RoboDK station: FanucComputerVisionSimulation_V1.rdk

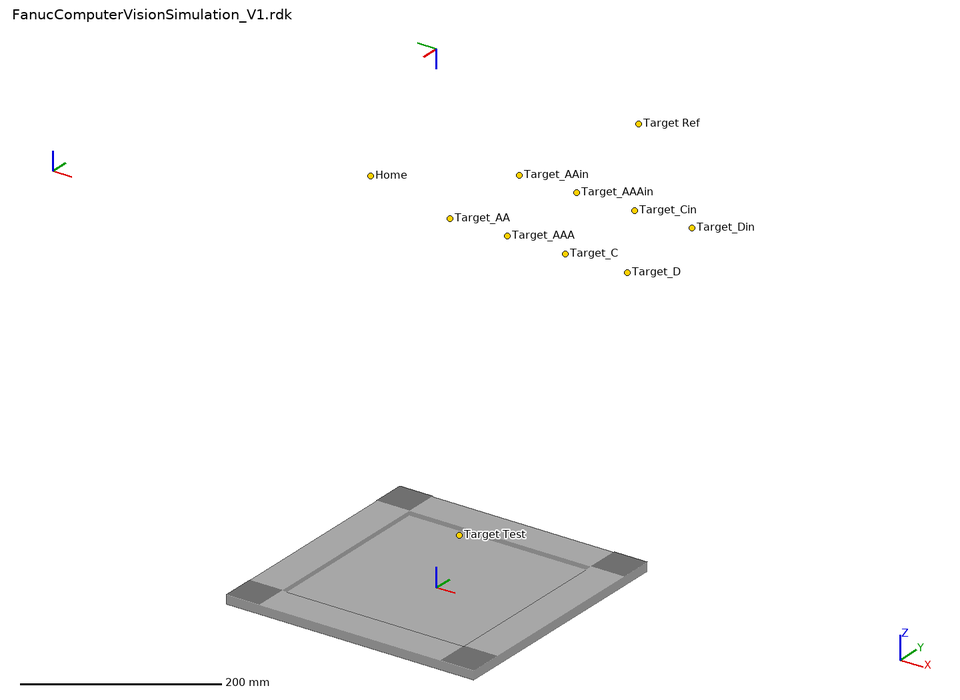
[picture v0: the station drawn from its stored meshes, robots at their saved joint values, targets as dots, program paths as lines]
Station FanucComputerVisionSimulation_V1 (saved by RoboDK 5.5.4). Poses are relative to the parent item; angles as X-Y-Z fixed-axis rotations.
Station parameters (name, value as stored): boardCenter, (319.0, 239.5, True), battery0, (496.821942952221, 61.274491474303716), battery1, (530.5798901508712, -36.737235512468814), battery2, (410.82767440352166, 59.47826360901432), battery3, (391.48109251529473, -70.56545100399168)
  - frame Fanuc LR Mate 200iD Base at (0, 0, 330) mm
    - robot Fanuc LR Mate 200iD: 6 axes, payload 7 kg, reach 717 mm, repeatability 0.02 mm, weight 25 kg
        modified DH rows (alpha deg, a mm, theta deg, d mm): 0, 0, 0, 330; -90, 50, -90, 0; 0, 330, 0, 0; -90, 35, 0, 335; 90, 0, 0, 0; -90, 0, 0, 80
        base shift (0, 0, -330) mm
        joint limits [-170, -100, -67, -190, -125, -360] to [170, 145, 213, 190, 125, 360]; home [0, 0, 0, 0, 0, 0]; saved at [0, 0, 0, 0, -90, 0]
      - frame My Camera Frame at (80, 0, 20) mm, rotated rx 0 ry 0 rz 90 deg
      - tool Gripper, TCP at (0, 0, 183) mm
    - frame Reference SW at (465, 0, -330) mm
      - object Work_Table at (0, 0, 0) mm, size 300 x 300 x 10 mm, 1061997773 curves, geometry from Flange_Holder.stl
        - object 4x4_1000-0 at (110, 110, 10.5) mm, size 40.5 x 40.5 x 0 mm, 862301904 curves, geometry from 4x4_1000-0.svg
        - object 4x4_1000-1 at (110, -150, 10.5) mm, size 40.5 x 40.5 x 0 mm, 862300704 curves, geometry from 4x4_1000-1.svg
        - object 4x4_1000-2 at (-150, -150, 10.5) mm, size 40.5 x 40.5 x 0 mm, 862301664 curves, geometry from 4x4_1000-2.svg
        - object 4x4_1000-3 at (-150, 110, 10.5) mm, size 40.5 x 40.5 x 0 mm, 862302864 curves, geometry from 4x4_1000-3.svg
      - target Home (Cartesian target) at (-80, 0, 432) mm, rotated rx -180 ry 0 rz 0 deg; joints [0, 0, 0, 0, -90, 0] of Fanuc LR Mate 200iD
      - target Target Ref (Cartesian target) at (70, 250, 432) mm, rotated rx -180 ry 0 rz 0 deg; joints [25.046, 43.834, 16.178, 0, -106.178, -25.046] of Fanuc LR Mate 200iD
      - target Target Test (Cartesian target) at (68.34, -58.43, 100) mm, rotated rx -180 ry 0 rz 0 deg; joints [7.615, 7.792, -3.745, 0, -86.255, -7.615] of Fanuc LR Mate 200iD
      - target Target_AA (Cartesian target) at (-110, 180, 305) mm, rotated rx -180 ry 0 rz 0 deg; joints [26.887, 3.808, -20.454, 0, -69.546, -26.887] of Fanuc LR Mate 200iD
      - target Target_AAA (Cartesian target) at (-40, 180, 305) mm, rotated rx -180 ry 0 rz 0 deg; joints [22.954, 14.574, -18.722, 0, -71.278, -22.954] of Fanuc LR Mate 200iD
      - target Target_C (Cartesian target) at (30, 180, 305) mm, rotated rx -180 ry 0 rz 0 deg; joints [19.983, 25.857, -14.839, 0, -75.161, -19.983] of Fanuc LR Mate 200iD
      - target Target_D (Cartesian target) at (105, 180, 305) mm, rotated rx -180 ry 0 rz 0 deg; joints [17.526, 39.754, -7.445, 0, -82.555, -17.526] of Fanuc LR Mate 200iD
      - target Target_AAin (Cartesian target) at (-110, 300, 305) mm, rotated rx -180 ry 0 rz 0 deg; joints [40.2, 15.123, -18.581, 0, -71.419, -40.2] of Fanuc LR Mate 200iD
      - target Target_AAAin (Cartesian target) at (-40, 300, 305) mm, rotated rx -180 ry 0 rz 0 deg; joints [35.218, 24.697, -15.33, 0, -74.67, -35.218] of Fanuc LR Mate 200iD
      - target Target_Cin (Cartesian target) at (30, 300, 305) mm, rotated rx -180 ry 0 rz 0 deg; joints [31.218, 35.742, -9.854, 0, -80.146, -31.218] of Fanuc LR Mate 200iD
      - target Target_Din (Cartesian target) at (100, 300, 305) mm, rotated rx -180 ry 0 rz 0 deg; joints [27.967, 50.525, 0.035, 0, -90.035, -27.967] of Fanuc LR Mate 200iD
  - Python program CameraProgram (listed below)
  - camera My Camera
  - object Table 108x114x32 IN at (-435, 0, -467.5) mm
  - Python program TakePhoto (listed below)
  - Python program SearchWorkArea (listed below)
  - Python program Test (listed below)
  - Python program CollectImages_size (listed below)
  - Python program CollectImages_brand (listed below)
  - frame Bateries at (-10000, 1500, 22) mm
    - object 9V(Duracell) at (0, 0, 0) mm
    - object 9V(Energizer) at (0, 0, 0) mm
    - object 9V(Lorem Ipsum) at (0, 0, 0) mm
    - object AA(Duracell) at (200, 0, -10) mm
    - object AA(Energizer) at (200, 80, -10) mm
    - object AA(Lorem Ipsum) at (200, 160, -10) mm
    - object AAA(Duracell) at (160, 0, -12) mm
    - object AAA(Energizer) at (160, 80, -12) mm
    - object AAA(Lorem Ipsum) at (160, 160, -12) mm
    - object C(Duracell) at (120, 0, -4) mm, size 6 x 3 x 6 mm, 1058642330 curves, geometry from C(Duracell).obj
    - object C(Energizer) at (120, 80, -4) mm, size 6 x 3 x 6 mm, 1058642330 curves, geometry from C(Energizer).obj
    - object C(Lorem Ipsum) at (120, 160, -4) mm, size 6 x 3 x 6 mm, 1058642330 curves, geometry from C(Lorem Ipsum).obj
    - object D(Duracell) at (80, 0, 0) mm, size 6 x 3 x 6 mm, 1058642330 curves, geometry from D(Duracell).obj
    - object D(Energizer) at (80, 80, 0) mm, size 6 x 3 x 6 mm, 1058642330 curves, geometry from D(Energizer).obj
    - object D(Lorem Ipsum) at (80, 160, 0) mm, size 6 x 3 x 6 mm, 1058642330 curves, geometry from D(Lorem Ipsum).obj
  - Python program Sort (listed below)
  - Python program SpawnObjects (listed below)
  - Python program DeleteObjects (listed below)
  - object Box at (465, 300, 0) mm

--- Python program CameraProgram ---
from robodk import robolink  # RoboDK API
from robodk import robomath  # Robot toolbox
RDK = robolink.Robolink()

import numpy as np
import cv2 as cv
import time

CAM_SIZE = 640, 480

CAM_NAME = 'My Camera'
CAM_PARAMS = f'SIZE={CAM_SIZE[0]}x{CAM_SIZE[1]}'
WINDOW_NAME = 'My Camera Feed'

boardCenter = (None, None, False)
def aruco_display(corners, ids, rejected, image):
    #Draw Middle Cross-Hair
    crossHair = 20
    cv.line(image, (CAM_SIZE[0]//2 - crossHair, CAM_SIZE[1]//2), (CAM_SIZE[0]//2 + crossHair, CAM_SIZE[1]//2), (255, 0, 0), 1)
    cv.line(image, (CAM_SIZE[0]//2, CAM_SIZE[1]//2 - crossHair), (CAM_SIZE[0]//2, CAM_SIZE[1]//2 + crossHair), (255, 0, 0), 1)

    #Check If Marker Present
    if len(corners) > 0:
        ids = ids.flatten()
        workCorners = [ #limits of work area
            [0, None],
            [1, None],
            [2, None],
            [3, None]
        ]

        #Catch All Markers
        for (markerCorner, markerID) in zip(corners, ids):
            corners = markerCorner.reshape((4, 2))
            (topRight, bottomRight, bottomLeft, topLeft) = corners

            topRight = (int(topRight[0]), int(topRight[1]))
            topLeft = (int(topLeft[0]), int(topLeft[1]))
            bottomRight = (int(bottomRight[0]), int(bottomRight[1]))
            bottomLeft= (int(bottomLeft[0]), int(bottomLeft[1]))

            cv.line(image, topLeft, topRight, (0, 255, 0), 2)
            cv.line(image, topRight, bottomRight, (0, 255, 0), 2)
            cv.line(image, bottomRight, bottomLeft, (0, 255, 0), 2)
            cv.line(image, bottomLeft, topLeft, (0, 255, 0), 2)

            match markerID:
                case 0:
                    dotPos = topLeft
                case 1:
                    dotPos = topRight
                case 2:
                    dotPos = bottomRight
                case 3:
                    dotPos = bottomLeft
            cv.circle(image, dotPos, 4, (0, 0, 255), -1)
            workCorners[markerID][1] = dotPos
            cv.putText(image, str(markerID), (int((topLeft[0] + bottomRight[0])/2.0), int((topLeft[1] + bottomRight[1])/2.0)), cv.FONT_HERSHEY_SIMPLEX, 0.5, (0, 0, 255), 2)

            centerFound = True
            global boardCenter
            for corner in workCorners:
                if corner[1] is None:
                    centerFound = False
                    break
            if centerFound:
                boardCenter = ((workCorners[0][1][0] + workCorners[2][1][0])/2.0, (workCorners[0][1][1] + workCorners[2][1][1])/2.0, True)
                print(boardCenter)
                cv.circle(image, (int(boardCenter[0]), int(boardCenter[1])), 10, (0, 0, 255), 2)
                cv.circle(image, (0, 0), 10, (0, 0, 255), 2)
            else:
                boardCenter = (None, None, False)

        #Draw Work Area
        for i in range(len(workCorners)):
            start_corner = workCorners[i][1]
            end_corner = workCorners[(i + 1) % len(workCorners)][1]
            if start_corner and end_corner is not None:
                cv.line(image, start_corner, end_corner, (0, 0, 255), 2)
    RDK.setParam('boardCenter', boardCenter)
    return image

#----------------------------------
# Get the camera item
cam_item = RDK.Item(CAM_NAME, robolink.ITEM_TYPE_CAMERA)
if not cam_item.Valid():
    cam_item = RDK.Cam2D_Add(RDK.AddFrame(CAM_NAME + ' Frame'), CAM_PARAMS)
    cam_item.setName(CAM_NAME)
cam_item.setParam('Open', 1)

#----------------------------------
# Aruco Setup
arucoType = "DICT_4x4_50"
arucoDict = cv.aruco.getPredefinedDictionary(cv.aruco.DICT_4X4_50)
arucoParams = cv.aruco.DetectorParameters()

#----------------------------------
# Create a live feed
while cam_item.setParam('isOpen') == '1':
    #----------------------------------
    # Method 1: Get the camera image, by socket
    img_socket = None
    bytes_img = RDK.Cam2D_Snapshot('', cam_item)
    if isinstance(bytes_img, bytes) and bytes_img != b'':
        nparr = np.frombuffer(bytes_img, np.uint8)
        img_socket = cv.imdecode(nparr, cv.IMREAD_COLOR)
    if img_socket is None:
        break

    corners, ids, rejected = cv.aruco.detectMarkers(img_socket, arucoDict, parameters=arucoParams)
    detected_markers = aruco_display(corners, ids, rejected, img_socket)

    #----------------------------------
    # Show it to the world!
    cv.imshow(WINDOW_NAME, detected_markers)

    key = cv.waitKey(1)
    if key == 27:
        break  # User pressed ESC, exit
    if cv.getWindowProperty(WINDOW_NAME, cv.WND_PROP_VISIBLE) < 1 and cv.getWindowProperty('Cropped', cv.WND_PROP_VISIBLE) < 1:
        break  # User killed the main window, exit

# Close the preview and the camera. Ensure you call cam_item.setParam('Open', 1) before reusing a camera!
cv.destroyAllWindows()
RDK.Cam2D_Close(cam_item)

--- Python program TakePhoto ---
# Type help("robodk.robolink") or help("robodk.robomath") for more information
# Press F5 to run the script
# Documentation: https://robodk.com/doc/en/RoboDK-API.html
# Reference:     https://robodk.com/doc/en/PythonAPI/robodk.html
# Note: It is not required to keep a copy of this file, your Python script is saved with your RDK project

# You can also use the new version of the API:
from robodk import robolink    # RoboDK API
from robodk import robomath    # Robot toolbox
RDK = robolink.Robolink()

# Forward and backwards compatible use of the RoboDK API:
# Remove these 2 lines to follow python programming guidelines
from robodk import *      # RoboDK API
from robolink import *    # Robot toolbox
# Link to RoboDK
# RDK = Robolink()

import cv2 as cv
import numpy as np

CAM_SIZE = 640, 480

CAM_NAME = 'My Camera'
CAM_PARAMS = f'SIZE={CAM_SIZE[0]}x{CAM_SIZE[1]}'
WINDOW_NAME = 'My Camera Feed'

# Get the camera item
cam_item = RDK.Item(CAM_NAME, robolink.ITEM_TYPE_CAMERA)
if not cam_item.Valid():
    cam_item = RDK.Cam2D_Add(RDK.AddFrame(CAM_NAME + ' Frame'), CAM_PARAMS)
    cam_item.setName(CAM_NAME)
cam_item.setParam('Open', 1)

screenshotCount = 8
# Create a live feed
while cam_item.setParam('isOpen') == '1':
    #----------------------------------
    # Method 1: Get the camera image, by socket
    img_socket = None
    bytes_img = RDK.Cam2D_Snapshot('', cam_item)
    if isinstance(bytes_img, bytes) and bytes_img != b'':
        nparr = np.frombuffer(bytes_img, np.uint8)
        img_socket = cv.imdecode(nparr, cv.IMREAD_COLOR)
    if img_socket is None:
        break

    crop_img = img_socket[69:409, 150:490]
    cv.imshow("Cropped", crop_img)
    if screenshotCount<100:
        screenshotCount += 1

        RDK.RunCode("PoseObjects", True)

        cv.imwrite(f'D:\L I C E N T A\Simulare\Training images\ImgToTrain_{screenshotCount}.jpg', crop_img)
        print(f'Image saves as: ImgToTrain_{screenshotCount}')

        RDK.RunCode("DeleteObjects", True)

    key = cv.waitKey(1)
    if key == 27:
        break  # User pressed ESC, exit
    if cv.getWindowProperty(WINDOW_NAME, cv.WND_PROP_VISIBLE) < 1 and cv.getWindowProperty('Cropped', cv.WND_PROP_VISIBLE) < 1:
        break  # User killed the main window, exit

# Close the preview and the camera. Ensure you call cam_item.setParam('Open', 1) before reusing a camera!
cv.destroyAllWindows()
RDK.Cam2D_Close(cam_item)

--- Python program SearchWorkArea ---
from robodk import robolink    # RoboDK API
from robodk import robomath    # Robot toolbox
RDK = robolink.Robolink()

from robodk import *      # RoboDK API
from robolink import *    # Robot toolbox

import math
import cv2 as cv
import threading

# Connect Robot Arm
robot = RDK.Item(r'Fanuc LR Mate 200iD')
if not robot.Valid():
    raise Exception('Robot not connected!')
robot.setPoseFrame(robot.PoseFrame())
robot.setPoseTool(robot.PoseTool())
robot.setRounding(10)
robot.setSpeed(25)

target_ref = robot.Pose()
pos_ref = target_ref.Pos()

accuracy = 1e-8

workArea_Found = False
def moveRobot(robot, targ_ref, point):
    current_target = Mat(targ_ref)
    current_pos = current_target.Pos()
    current_pos[0] += point[0]
    current_pos[1] += point[1]
    current_target.setPos(current_pos)
    robot.MoveL(current_target)
def searchWork(searchArea):
    dirX = 1
    dirY = 1
    for i in range(segments*2):
        workArea_Find()
        current_target = robot.Pose()
        current_pos = Mat(current_target).Pos()

        dirY = 1 if i>=segments else -1

        next_point = (0, searchArea[1]*dirY/segments)
        moveRobot(robot, current_target, next_point)

        current_target = robot.Pose()
        current_pos = Mat(current_target).Pos()

        dirX = -dirX

        next_point = (searchArea[0]*dirX, 0)
        moveRobot(robot, current_target, next_point)
def workArea_Find():
    global workArea_Found
    counter = 0
    while True:
        counter += 1
        print(f"Frame: {counter}")
        boardCenter = RDK.getParam('boardCenter')
        if boardCenter[2]:
            print("Detected")
            robot.Stop()
def moveRobotJoints(speed):
    move_direction = (0, 0, 0)

start_point = 150, 250
end_point = -150, -250

searchArea = (start_point[0] - end_point[0]), (start_point[1] - end_point[1])

directionX = 1
directionY = 1
segments = 10

moveRobot(robot, target_ref, start_point)

findWork_thread = threading.Thread(target=workArea_Find)
findWork_thread.start()

while True:
    searchWork(searchArea)
    key = cv.waitKey(1)
    if key == 27 and workArea_Found:
            break  # User pressed ESC, exit

--- Python program Test ---
from robodk.robolink import *  # API to communicate with RoboDK
from robodk.robomath import *  # basic matrix operations

RDK = Robolink()

# Arrow keys program example

# get a robot
robot = RDK.Item('', ITEM_TYPE_ROBOT)
if not robot.Valid():
    print("No robot in the station. Load a robot first, then run this program.")
    pause(5)
    raise Exception("No robot in the station!")

print('Using robot: %s' % robot.Name())
print('Use the arrows (left, right, up, down), Q and A keys to move the robot')
print('Note: This works on console mode only, you must run the PY file separately')

# define the move increment
move_speed = 1

from msvcrt import getch

while True:
    #key = (ord(getch()))
    move_direction = [0, 0, 0]
    key = 97
    if key == 75:
        print('arrow left (Y-)')
        move_direction = [0, -1, 0]
    elif key == 77:
        print('arrow right (Y+)')
        move_direction = [0, 1, 0]
    elif key == 72:
        print('arrow up (X-)')
        move_direction = [-1, 0, 0]
    elif key == 80:
        print('arrow down (X+)')
        move_direction = [1, 0, 0]
    elif key == 113:
        print('Q (Z+)')
        move_direction = [0, 0, 1]
    elif key == 97:
        print('A (Z-)')
        move_direction = [0, 0, -1]

    # make sure that a movement direction is specified
    if norm(move_direction) <= 0:
        continue

    # calculate the movement in mm according to the movement speed
    xyz_move = mult3(move_direction, move_speed)

    # get the robot joints
    robot_joints = robot.Joints()

    # get the robot position from the joints (calculate forward kinematics)
    robot_position = robot.SolveFK(robot_joints)
    print(robot_position)

    # get the robot configuration (robot joint state)
    robot_config = robot.JointsConfig(robot_joints)

    # calculate the new robot position
    new_robot_position = transl(xyz_move) * robot_position

    # calculate the new robot joints
    new_robot_joints = robot.SolveIK(new_robot_position)
    if len(new_robot_joints.tolist()) < 6:
        print("No robot solution!! The new position is too far, out of reach or close to a singularity")
        continue

    # calculate the robot configuration for the new joints
    new_robot_config = robot.JointsConfig(new_robot_joints)

    # if robot_config[0] != new_robot_config[0] or robot_config[1] != new_robot_config[1] or robot_config[2] != new_robot_config[2]:
    #     print("Warning!! Robot configuration changed!! This will lead to unextected movements!")
    #     print(robot_config)
    #     print(new_robot_config)

        # move the robot joints to the new position
    robot.MoveJ(new_robot_joints)
        #robot.MoveL(new_robot_joints)

--- Python program CollectImages_size ---
from robodk import robolink    # RoboDK API
from robodk import robomath    # Robot toolbox
RDK = robolink.Robolink()

import random
import math
import cv2 as cv
import numpy as np
import os

battery_names_list = [
    'AA(Duracell)', 'AA(Energizer)', 'AA(Lorem Ipsum)',
    'AAA(Duracell)', 'AAA(Energizer)', 'AAA(Lorem Ipsum)',
    'C(Duracell)', 'C(Energizer)', 'C(Lorem Ipsum)',
    'D(Duracell)', 'D(Energizer)', 'D(Lorem Ipsum)'
]
battery_sizes = [
    (0, 'AA', 52.5, 16.5),
    (1, 'AAA', 46.5, 12.5),
    (2, 'C', 52, 28.2),
    (3, 'D', 63.5, 36.2)
]
spaws_limits = [
    [(495, 540), (35, 75)],
    [(495, 540), (-75, -35)],
    [(390, 435), (35, 75)],
    [(390, 435), (-75, -35)]
]

battery = {}
copy = {}

CAM_SIZE = 640, 480
MM_2_PIX = 340/220

CAM_NAME = 'My Camera'
CAM_PARAMS = f'SIZE={CAM_SIZE[0]}x{CAM_SIZE[1]}'
WINDOW_NAME = 'My Camera Feed'

cam_item = RDK.Item(CAM_NAME, robolink.ITEM_TYPE_CAMERA)
if not cam_item.Valid():
    cam_item = RDK.Cam2D_Add(RDK.AddFrame(CAM_NAME + ' Frame'), CAM_PARAMS)
    cam_item.setName(CAM_NAME)
cam_item.setParam('Open', 1)

screenshotCount = 0
table_origin = 575, 110
box_data = {}
# Retrieve objects by name and store them in the dictionary
for name in battery_names_list:
    obj = RDK.Item(name, robolink.ITEM_TYPE_OBJECT)
    if obj.Valid():
        battery[name] = obj
    else:
        print(f"{name} not found!")

# Check if any valid objects were found
if not battery:
    print("No valid objects found!")

def boxSize(angle, x, y, width, height):
    width *= MM_2_PIX
    height *= MM_2_PIX
    theta = angle
    deg_angle = math.degrees(angle)
    cos_theta = math.cos(theta)
    sin_theta = math.sin(theta)

    # Calculate the coordinates of the corners of the rotated rectangle
    x_min = x - width / 2
    y_min = y - height / 2
    x_max = x + width / 2
    y_max = y + height / 2

    corner = [[0, 0] for _ in range(4)]
    corner[0][0] = x + cos_theta * (x_min - x) - sin_theta * (y_min - y)
    corner[0][1] = y + sin_theta * (x_min - x) + cos_theta * (y_min - y)

    corner[2][0] = x + cos_theta * (x_max - x) - sin_theta * (y_max - y)
    corner[2][1] = y + sin_theta * (x_max - x) + cos_theta * (y_max - y)

    corner[1][0] = x + cos_theta * (x_min - x) - sin_theta * (y_max- y)
    corner[1][1] = y + sin_theta * (x_min - x) + cos_theta * (y_max - y)

    corner[3][0] = x + cos_theta * (x_max - x) - sin_theta * (y_min - y)
    corner[3][1] = y + sin_theta * (x_max - x) + cos_theta * (y_min - y)

    all_x = [c[0] for c in corner]
    all_y = [c[1] for c in corner]

    x_min = min(all_x)
    y_min = min(all_y)
    x_max = max(all_x)
    y_max = max(all_y)

    new_height = x_max - x_min
    new_width = y_max - y_min

    return new_width, new_height

def convertYolo(image_width, image_height, x, y, boxW, boxH):
    x_center = x/image_width
    y_center = y/image_height
    box_width = boxW/image_width
    box_height = boxH/image_height

    return (x_center, y_center, box_width, box_height)
def createLabel(type, x, y, boxW, boxH):
    filename = f"D:/L I C E N T A/Simulare/Training Images/Data/Size/Labels/ImgToTrain_{screenshotCount+1}.txt"
    if os.path.exists(filename):
        with open(filename, 'r') as file:
            lines = file.readlines()

        if len(lines) >= 4:
            mode = 'w'
        else:
            mode = 'a'
    else:
        mode = 'w'

    with open(filename, mode) as file:
        file.write(f"{type} {round(x, 5)} {round(y, 5)} {round(boxW, 5)} {round(boxH, 5)}" + '\n')
def spawnNewBatteries(img):
    global battery
    global copy
    global box
    for i in range(4):
        random_battery = random.choice(list(battery.keys()))
        battery[random_battery].Copy()
        copy[i] = RDK.Paste()

        random_pose = battery[random_battery].PoseAbs()

        random_x = random.uniform(spaws_limits[i][0][0], spaws_limits[i][0][1])
        random_y = random.uniform(spaws_limits[i][1][0], spaws_limits[i][1][1])
        random_angle_y = math.radians(random.uniform(0, 360))  # Random angle around Y axis
        random_angle_z = math.radians(random.uniform(0, 360))  # Random angle around Z axis
        transl_matrix = robomath.transl(random_x, random_y, random_pose[2, 3]) * robomath.rotz(random_angle_z) * robomath.roty(random_angle_y)

        copy[i].setPoseAbs(transl_matrix)
        copy[i].setName(copy[i].Name() + '_COPY')

        copy_type = copy[i].Name()[:copy[i].Name().find("(")]

        #Reversed X and Y, the orientation of the robot is diferent
        boxY = (table_origin[0] - random_x) * MM_2_PIX
        boxX = (table_origin[1] - random_y) * MM_2_PIX

        for battery_data in battery_sizes:
            if battery_data[1] == copy_type:
                kind, _, h, w = battery_data
                boxH, boxW = boxSize(random_angle_z, boxX, boxY, h, w)
                yoloX, yoloY, yoloW, yoloH = convertYolo(340, 340, boxX, boxY, boxW, boxH)
                createLabel(kind, yoloX, yoloY, yoloW, yoloH)

                box_data[i] = (boxX, boxY, boxW, boxH)
                break

def deleteSpawnedBatteries():
    global copy
    for i in range(4):
        copy[i].Delete()

takePhoto = False
while cam_item.setParam('isOpen') == '1':
    img_socket = None
    bytes_img = RDK.Cam2D_Snapshot('', cam_item)
    if isinstance(bytes_img, bytes) and bytes_img != b'':
        nparr = np.frombuffer(bytes_img, np.uint8)
        img_socket = cv.imdecode(nparr, cv.IMREAD_COLOR)
    if img_socket is None:
        break

    crop_img = img_socket[69:409, 150:490]
    cv.imshow("Cropped", crop_img)

    if screenshotCount<100:

        if takePhoto:
            deleteSpawnedBatteries()
            box = box_data
            # for i in range(4):
            #     cv.circle(crop_img, [int(box[i][0]), int(box[i][1])], radius=1, color = (0, 0, 255), thickness=-1)
            #     cv.rectangle(crop_img, [int(box[i][0]-box[i][2]/2), int(box[i][1]-box[i][3]/2)], [int(box[i][0]+box[i][2]/2), int(box[i][1]+box[i][3]/2)], (0, 255, 0), 2)
        else:
            takePhoto = True
        cv.waitKey(500)

        spawnNewBatteries(crop_img)
        cv.waitKey(500)

        cv.imshow("Cropped", crop_img)
        cv.imwrite(f'D:/L I C E N T A/Simulare/Training Images/Data/Size/Images/ImgToTrain_{screenshotCount}.jpg', crop_img)

        print(f'Image saves as: ImgToTrain_{screenshotCount}')
        screenshotCount += 1

    key = cv.waitKey(1)
    if key == 27:
        break  # User pressed ESC, exit
    if cv.getWindowProperty(WINDOW_NAME, cv.WND_PROP_VISIBLE) < 1 and cv.getWindowProperty('Cropped', cv.WND_PROP_VISIBLE) < 1 or screenshotCount == 1000:
        deleteSpawnedBatteries()
        break  # User killed the main window, exit

# Close the preview and the camera. Ensure you call cam_item.setParam('Open', 1) before reusing a camera!
cv.destroyAllWindows()
RDK.Cam2D_Close(cam_item)

--- Python program CollectImages_brand ---
from robodk import robolink    # RoboDK API
from robodk import robomath    # Robot toolbox
RDK = robolink.Robolink()

import random
import math
import cv2 as cv
import numpy as np
import os

# Initialize the RoboDK API
RDK = robolink.Robolink()

# List of object names
battery_names_list = [
    'AA(Duracell)', 'AA(Energizer)', 'AA(Lorem Ipsum)',
    'AAA(Duracell)', 'AAA(Energizer)', 'AAA(Lorem Ipsum)',
    'C(Duracell)', 'C(Energizer)', 'C(Lorem Ipsum)',
    'D(Duracell)', 'D(Energizer)', 'D(Lorem Ipsum)'
]
battery_sizes= [
    (0, 'AA', 52.5, 16.5),
    (1, 'AAA', 46.5, 12.5),
    (2, 'C', 52, 28.2),
    (3, 'D', 63.5, 36.2)
]
battery_types= [
    (0, 'Duracell'),
    (1, 'Energizer'),
    (2, 'Lorem Ipsum')
]
spaws_limits = [
    [(495, 540), (35, 75)],
    [(495, 540), (-75, -35)],
    [(390, 435), (35, 75)],
    [(390, 435), (-75, -35)]
]
# Dictionary to store the original objects and their copies
battery = {}
copy = {}

CAM_SIZE = 640, 480
MM_2_PIX = 340/220

CAM_NAME = 'My Camera'
CAM_PARAMS = f'SIZE={CAM_SIZE[0]}x{CAM_SIZE[1]}'
WINDOW_NAME = 'My Camera Feed'

# Get the camera item
cam_item = RDK.Item(CAM_NAME, robolink.ITEM_TYPE_CAMERA)
if not cam_item.Valid():
    cam_item = RDK.Cam2D_Add(RDK.AddFrame(CAM_NAME + ' Frame'), CAM_PARAMS)
    cam_item.setName(CAM_NAME)
cam_item.setParam('Open', 1)

screenshotCount = 2501
table_origin = 575, 110
box_data = {}
# Retrieve objects by name and store them in the dictionary
for name in battery_names_list:
    obj = RDK.Item(name, robolink.ITEM_TYPE_OBJECT)
    if obj.Valid():
        battery[name] = obj
    else:
        print(f"{name} not found!")

# Check if any valid objects were found
if not battery:
    print("No valid objects found!")

def boxSize(angle, x, y, width, height):
    width *= MM_2_PIX
    height *= MM_2_PIX
    theta = angle
    deg_angle = math.degrees(angle)
    cos_theta = math.cos(theta)
    sin_theta = math.sin(theta)

    # Calculate the coordinates of the corners of the rotated rectangle
    x_min = x - width / 2
    y_min = y - height / 2
    x_max = x + width / 2
    y_max = y + height / 2

    corner = [[0, 0] for _ in range(4)]
    corner[0][0] = x + cos_theta * (x_min - x) - sin_theta * (y_min - y)
    corner[0][1] = y + sin_theta * (x_min - x) + cos_theta * (y_min - y)

    corner[2][0] = x + cos_theta * (x_max - x) - sin_theta * (y_max - y)
    corner[2][1] = y + sin_theta * (x_max - x) + cos_theta * (y_max - y)

    corner[1][0] = x + cos_theta * (x_min - x) - sin_theta * (y_max- y)
    corner[1][1] = y + sin_theta * (x_min - x) + cos_theta * (y_max - y)

    corner[3][0] = x + cos_theta * (x_max - x) - sin_theta * (y_min - y)
    corner[3][1] = y + sin_theta * (x_max - x) + cos_theta * (y_min - y)

    all_x = [c[0] for c in corner]
    all_y = [c[1] for c in corner]

    x_min = min(all_x)
    y_min = min(all_y)
    x_max = max(all_x)
    y_max = max(all_y)

    new_height = x_max - x_min
    new_width = y_max - y_min

    return new_width, new_height

def convertYolo(image_width, image_height, x, y, boxW, boxH):
    x_center = x/image_width
    y_center = y/image_height
    box_width = boxW/image_width
    box_height = boxH/image_height

    return (x_center, y_center, box_width, box_height)
def createLabel(type, x, y, boxW, boxH):
    # Specify the file name
    filename = f"D:/L I C E N T A/Simulare/Training Images/Data/Brand/Labels/ImgToTrain_{screenshotCount+1}.txt"
    if os.path.exists(filename):
        # Read the file and count the number of rows
        with open(filename, 'r') as file:
            lines = file.readlines()

        if len(lines) >= 4:
            # If there are 4 or more rows, replace the content
            mode = 'w'
        else:
            # If there are fewer than 4 rows, append to the content
            mode = 'a'
    else:
        # If the file doesn't exist, create it and write to it
        mode = 'w'

    # Open the file in the determined mode
    with open(filename, mode) as file:
        file.write(f"{type} {round(x, 5)} {round(y, 5)} {round(boxW, 5)} {round(boxH, 5)}" + '\n')
def spawnNewBatteries(img):
    global battery
    global copy
    global box
    for i in range(4):
        random_battery = random.choice(list(battery.keys()))
        battery[random_battery].Copy()
        copy[i] = RDK.Paste()

        random_pose = battery[random_battery].PoseAbs()

        random_x = random.uniform(spaws_limits[i][0][0], spaws_limits[i][0][1])
        random_y = random.uniform(spaws_limits[i][1][0], spaws_limits[i][1][1])
        random_angle_y = math.radians(random.uniform(0, 360))  # Random angle around Y axis
        random_angle_z = math.radians(random.uniform(0, 360))  # Random angle around Z axis
        transl_matrix = robomath.transl(random_x, random_y, random_pose[2, 3]) * robomath.rotz(random_angle_z) * robomath.roty(random_angle_y)

        copy[i].setPoseAbs(transl_matrix)
        copy[i].setName(copy[i].Name() + '_COPY')

        copy_size = copy[i].Name()[:copy[i].Name().find("(")]
        copy_type = copy[i].Name()[copy[i].Name().find("(")+1:copy[i].Name().find(")")]
        print(copy_type)

        #Reversed X and Y, the orientation of the robot is diferent
        boxY = (table_origin[0] - random_x) * MM_2_PIX
        boxX = (table_origin[1] - random_y) * MM_2_PIX

        for battery_data in battery_sizes:
            if battery_data[1] == copy_size:
                for battery_brand in battery_types:
                    if battery_brand[1] == copy_type:
                        _, _, h, w = battery_data
                        kind, _ = battery_brand
                        boxH, boxW = boxSize(random_angle_z, boxX, boxY, h, w)
                        yoloX, yoloY, yoloW, yoloH = convertYolo(340, 340, boxX, boxY, boxW, boxH)
                        createLabel(kind, yoloX, yoloY, yoloW, yoloH)

                        box_data[i] = (boxX, boxY, boxW, boxH)
                break

def deleteSpawnedBatteries():
    global copy
    for i in range(4):
        copy[i].Delete()

takePhoto = False
while cam_item.setParam('isOpen') == '1':
    #----------------------------------
    # Method 1: Get the camera image, by socket
    img_socket = None
    bytes_img = RDK.Cam2D_Snapshot('', cam_item)
    if isinstance(bytes_img, bytes) and bytes_img != b'':
        nparr = np.frombuffer(bytes_img, np.uint8)
        img_socket = cv.imdecode(nparr, cv.IMREAD_COLOR)
    if img_socket is None:
        break

    crop_img = img_socket[69:409, 150:490]
    cv.imshow("Cropped", crop_img)

    if screenshotCount<2502:

        if takePhoto:
            deleteSpawnedBatteries()
            box = box_data
            # for i in range(4):
            #     cv.circle(crop_img, [int(box[i][0]), int(box[i][1])], radius=1, color = (0, 0, 255), thickness=-1)
            #     cv.rectangle(crop_img, [int(box[i][0]-box[i][2]/2), int(box[i][1]-box[i][3]/2)], [int(box[i][0]+box[i][2]/2), int(box[i][1]+box[i][3]/2)], (0, 255, 0), 2)
        else:
            takePhoto = True
        cv.waitKey(500)

        spawnNewBatteries(crop_img)
        cv.waitKey(500)

        cv.imshow("Cropped", crop_img)
        cv.imwrite(f'D:/L I C E N T A/Simulare/Training Images/Data/Brand/Images/ImgToTrain_{screenshotCount}.jpg', crop_img)

        print(f'Image saves as: ImgToTrain_{screenshotCount}')
        screenshotCount += 1

    key = cv.waitKey(1)
    if key == 27:
        break  # User pressed ESC, exit
    if cv.getWindowProperty(WINDOW_NAME, cv.WND_PROP_VISIBLE) < 1 and cv.getWindowProperty('Cropped', cv.WND_PROP_VISIBLE) < 1 or screenshotCount == 2501:
        deleteSpawnedBatteries()
        break  # User killed the main window, exit

# Close the preview and the camera. Ensure you call cam_item.setParam('Open', 1) before reusing a camera!
cv.destroyAllWindows()
RDK.Cam2D_Close(cam_item)

--- Python program Sort ---
from robodk import robolink    # RoboDK API
from robodk import robomath    # Robot toolbox
RDK = robolink.Robolink()

from robodk import *      # RoboDK API
from robolink import *    # Robot toolbox
# Link to RoboDK
# RDK = Robolink()

import os
from ultralytics import YOLO
import cv2 as cv
import numpy as np

CAM_SIZE = 640, 480

CAM_NAME = 'My Camera'
CAM_PARAMS = f'SIZE={CAM_SIZE[0]}x{CAM_SIZE[1]}'
WINDOW_NAME = 'My Camera Feed'
PIX_2_MM = 220/340

robot = RDK.Item(r'Fanuc LR Mate 200iD')
if not robot.Valid():
    raise Exception('Robot not connected!')

tool = RDK.Item("Gripper", robolink.ITEM_TYPE_TOOL)
robot.setPoseFrame(robot.PoseFrame())
robot.setPoseTool(robot.PoseTool())
robot.setRounding(10)
robot.setSpeed(10)

target_ref = robot.Pose()
pos_ref = target_ref.Pos()
abovePick_Z = 100
table_origin = 365, 110
offset = 10, 25

cam_item = RDK.Item(CAM_NAME, robolink.ITEM_TYPE_CAMERA)
if not cam_item.Valid():
    cam_item = RDK.Cam2D_Add(RDK.AddFrame(CAM_NAME + ' Frame'), CAM_PARAMS)
    cam_item.setName(CAM_NAME)
cam_item.setParam('Open', 1)

target_item = RDK.Item("Target Test", robolink.ITEM_TYPE_TARGET)
target_home = RDK.Item("Home", robolink.ITEM_TYPE_TARGET)
target_item.setPose(target_home.Pose())

target_AA = RDK.Item("Target_AA", robolink.ITEM_TYPE_TARGET)
target_AAA = RDK.Item("Target_AAA", robolink.ITEM_TYPE_TARGET)
target_C = RDK.Item("Target_C", robolink.ITEM_TYPE_TARGET)
target_D = RDK.Item("Target_D", robolink.ITEM_TYPE_TARGET)

target_AAin = RDK.Item("Target_AAin", robolink.ITEM_TYPE_TARGET)
target_AAAin = RDK.Item("Target_AAAin", robolink.ITEM_TYPE_TARGET)
target_Cin = RDK.Item("Target_Cin", robolink.ITEM_TYPE_TARGET)
target_Din = RDK.Item("Target_Din", robolink.ITEM_TYPE_TARGET)

targets_sort = [target_AA, target_AAA, target_C, target_D]
targets_sortIN = [target_AAin, target_AAAin, target_Cin, target_Din]

spawnBatteries = RDK.Item("SpawnObjects", robolink.ITEM_TYPE_PROGRAM_PYTHON)
deleteBatteries = RDK.Item("DeleteObjects", robolink.ITEM_TYPE_PROGRAM_PYTHON)

modelAI_path = "D:/L I C E N T A/Simulare/Scripts/YOLOv8_Model_Detection/generations/gen_5.pt"
modelAI = YOLO(modelAI_path)
threshold = 0.9

def convertCoordinates(x, y):
    new_x = table_origin[0] + x * PIX_2_MM + offset[0]
    new_y = table_origin[1] - y * PIX_2_MM - offset[1]
    return new_x, new_y

def getZ (class_id):
    battery_sizes = [
    ('AA', 16.5),
    ('AAA', 12.5),
    ('C', 28.2),
    ('D', 36.2)
    ]
    height = battery_sizes[class_id][1]
    return height

frame_placeHolder = np.zeros((100,100,3), dtype=np.uint8)
delayFrames = 60
frames = delayFrames
while cam_item.setParam('isOpen') == '1':
    img_socket = None
    bytes_img = RDK.Cam2D_Snapshot('', cam_item)
    if isinstance(bytes_img, bytes) and bytes_img != b'':
        nparr = np.frombuffer(bytes_img, np.uint8)
        img_socket = cv.imdecode(nparr, cv.IMREAD_COLOR)
    if img_socket is None:
        break

    frame_cut = img_socket[69:409, 150:490]
    frame = cv.rotate(frame_cut, cv.ROTATE_90_CLOCKWISE)

    scanResults = modelAI(frame, verbose=False)[0]

    robot_joints = robot.Joints()
    robot_position = robot.SolveFK(robot_joints)
    robot_config = robot.JointsConfig(robot_joints)

    for i, result in enumerate(scanResults.boxes.data.tolist()):
        x, y, w, h, score, class_id = result
        realX, realY = convertCoordinates(x, y)
        print(class_id ,realX, realY)
        target = (realX, realY, abovePick_Z)

        target_pose = target_item.PoseAbs()
        target_pose.setPos([realX, realY, abovePick_Z])
        target_item.setPoseAbs(target_pose)

        if score > threshold:
            cv.rectangle(frame, (int(x), int(y)), (int(w), int(h)), (0, 255, 0), 4)
            cv.putText(frame, scanResults.names[int(class_id)].upper(), (int(x), int(y - 10)), cv.FONT_HERSHEY_SIMPLEX, 0.8, (0, 255, 0), 1, cv.LINE_AA)
            cv.imshow(WINDOW_NAME, frame)
            robot.MoveL(target_item, blocking=True)
            cv.waitKey(1000)

            target_pose.setPos([realX, realY, getZ(int(class_id))])
            target_item.setPoseAbs(target_pose)
            robot.MoveL(target_item, blocking=True)
            tool.AttachClosest()
            cv.waitKey(1000)

            target_pose.setPos([realX, realY, abovePick_Z])
            target_item.setPoseAbs(target_pose)
            robot.MoveL(target_item, blocking=True)
            cv.waitKey(1000)

            currentTarget = targets_sort[int(class_id)]
            robot.MoveL(currentTarget, blocking=True)
            cv.waitKey(1000)

            currentTarget = targets_sortIN[int(class_id)]
            robot.MoveL(currentTarget, blocking=True)
            tool.DetachAll()
            cv.waitKey(1000)

            currentTarget = targets_sort[int(class_id)]
            robot.MoveL(currentTarget, blocking=True)
            cv.waitKey(1000)

            if i == len(scanResults.boxes.data.tolist())-1:
                deleteBatteries.RunProgram()
                spawnBatteries.RunProgram()
            cv.waitKey(3000)

            currentTarget = target_home
            robot.MoveL(currentTarget, blocking=True)
            cv.waitKey(1000)

    key = cv.waitKey(1)
    if key == 27:
        break  # User pressed ESC, exit
    if cv.getWindowProperty(WINDOW_NAME, cv.WND_PROP_VISIBLE) < 1 and cv.getWindowProperty('My Camera Feed', cv.WND_PROP_VISIBLE) < 1:
        break  # User killed the main window, exit

# Close the preview and the camera. Ensure you call cam_item.setParam('Open', 1) before reusing a camera!
cv.destroyAllWindows()
RDK.Cam2D_Close(cam_item)

--- Python program SpawnObjects ---
from robodk import robolink    # RoboDK API
from robodk import robomath    # Robot toolbox
RDK = robolink.Robolink()

# Forward and backwards compatible use of the RoboDK API:
# Remove these 2 lines to follow python programming guidelines
from robodk import *      # RoboDK API
from robolink import *    # Robot toolbox
# Link to RoboDK
# RDK = Robolink()
import random

battery_names_list = [
    'AA(Duracell)', 'AA(Energizer)', 'AA(Lorem Ipsum)',
    'AAA(Duracell)', 'AAA(Energizer)', 'AAA(Lorem Ipsum)',
    'C(Duracell)', 'C(Energizer)', 'C(Lorem Ipsum)',
    'D(Duracell)', 'D(Energizer)', 'D(Lorem Ipsum)'
]
spaws_limits = [
    [(495, 540), (35, 75)],
    [(495, 540), (-75, -35)],
    [(390, 435), (35, 75)],
    [(390, 435), (-75, -35)]
]
battery = {}
copy = {}

for name in battery_names_list:
    obj = RDK.Item(name, robolink.ITEM_TYPE_OBJECT)
    if obj.Valid():
        battery[name] = obj
    else:
        print(f"{name} not found!")

# Check if any valid objects were found
if not battery:
    raise("No valid objects found!")

def spawnNewBatteries():
    global battery
    global copy
    global box
    for i in range(4):
        random_battery = random.choice(list(battery.keys()))
        battery[random_battery].Copy()
        copy[i] = RDK.Paste()

        random_pose = battery[random_battery].PoseAbs()

        random_x = random.uniform(spaws_limits[i][0][0], spaws_limits[i][0][1])
        random_y = random.uniform(spaws_limits[i][1][0], spaws_limits[i][1][1])
        random_angle_y = math.radians(random.uniform(0, 360))  # Random angle around Y axis
        random_angle_z = math.radians(random.uniform(0, 360))  # Random angle around Z axis
        transl_matrix = robomath.transl(random_x, random_y, random_pose[2, 3]) * robomath.rotz(random_angle_z) * robomath.roty(random_angle_y)

        copy[i].setPoseAbs(transl_matrix)
        copy[i].setName(copy[i].Name() + '_COPY')


spawnNewBatteries()

--- Python program DeleteObjects ---
# Type help("robodk.robolink") or help("robodk.robomath") for more information
# Press F5 to run the script
# Documentation: https://robodk.com/doc/en/RoboDK-API.html
# Reference:     https://robodk.com/doc/en/PythonAPI/robodk.html
# Note: It is not required to keep a copy of this file, your Python script is saved with your RDK project

# You can also use the new version of the API:
from robodk import robolink    # RoboDK API
from robodk import robomath    # Robot toolbox
RDK = robolink.Robolink()

# Forward and backwards compatible use of the RoboDK API:
# Remove these 2 lines to follow python programming guidelines
from robodk import *      # RoboDK API
from robolink import *    # Robot toolbox

RDK = robolink.Robolink()

# Get all items in the station
all_items = RDK.ItemList()

# Define the substring to search for
substring = "_COPY"

# Filter items that contain the substring
filtered_items = [item for item in all_items if substring in item.Name()]

# Print the names of the filtered items
for item in filtered_items:
    item.Delete()
